FUNCTION_BLOCK FB_CheckAnyMode
VAR_INPUT
	
stn1:FB_Mode;
stn2:FB_Mode;
stn3:FB_Mode;
stn4:FB_Mode;
stn5:FB_Mode;
stn6:FB_Mode;


END_VAR
VAR_OUTPUT
	LockedModes:typeStationLockModes;
END_VAR
VAR
	tAnyAutoMode: BOOL;
	tAnyManualMode: BOOL;
END_VAR

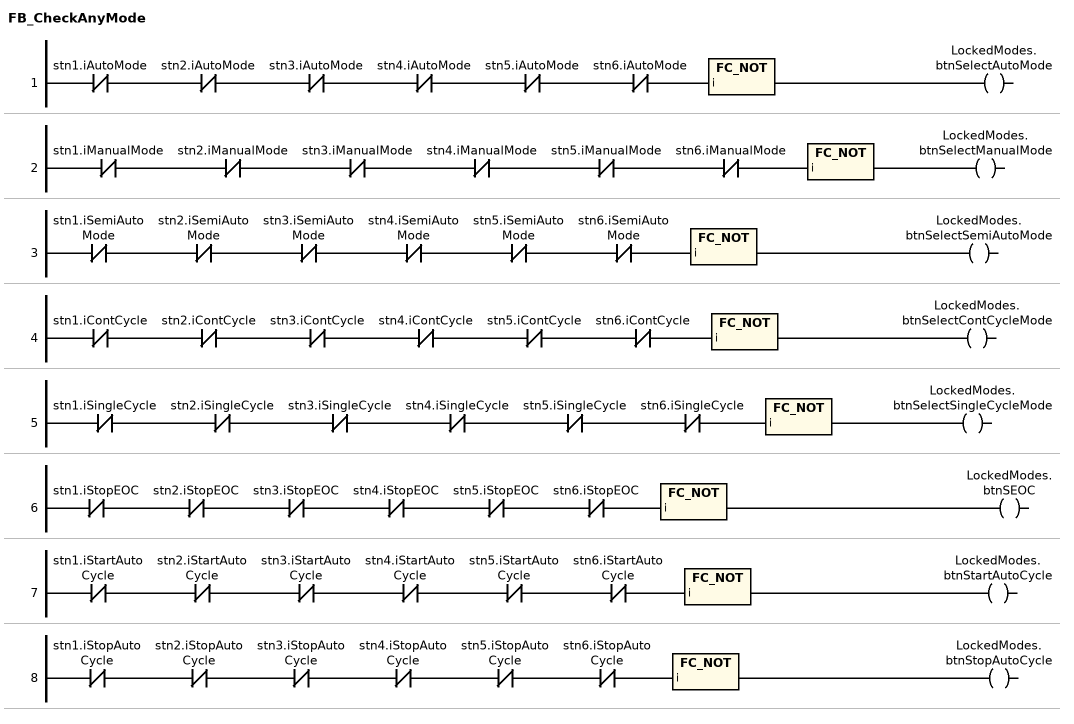
// NETWORK 1
LockedModes.btnSelectAutoMode := FC_NOT(i := NOT stn1.iAutoMode AND NOT stn2.iAutoMode AND NOT stn3.iAutoMode AND NOT stn4.iAutoMode AND NOT stn5.iAutoMode AND NOT stn6.iAutoMode);

// NETWORK 2
LockedModes.btnSelectManualMode := FC_NOT(i := NOT stn1.iManualMode AND NOT stn2.iManualMode AND NOT stn3.iManualMode AND NOT stn4.iManualMode AND NOT stn5.iManualMode AND NOT stn6.iManualMode);

// NETWORK 3
LockedModes.btnSelectSemiAutoMode := FC_NOT(i := NOT stn1.iSemiAutoMode AND NOT stn2.iSemiAutoMode AND NOT stn3.iSemiAutoMode AND NOT stn4.iSemiAutoMode AND NOT stn5.iSemiAutoMode AND NOT stn6.iSemiAutoMode);

// NETWORK 4
LockedModes.btnSelectContCycleMode := FC_NOT(i := NOT stn1.iContCycle AND NOT stn2.iContCycle AND NOT stn3.iContCycle AND NOT stn4.iContCycle AND NOT stn5.iContCycle AND NOT stn6.iContCycle);

// NETWORK 5
LockedModes.btnSelectSingleCycleMode := FC_NOT(i := NOT stn1.iSingleCycle AND NOT stn2.iSingleCycle AND NOT stn3.iSingleCycle AND NOT stn4.iSingleCycle AND NOT stn5.iSingleCycle AND NOT stn6.iSingleCycle);

// NETWORK 6
LockedModes.btnSEOC := FC_NOT(i := NOT stn1.iStopEOC AND NOT stn2.iStopEOC AND NOT stn3.iStopEOC AND NOT stn4.iStopEOC AND NOT stn5.iStopEOC AND NOT stn6.iStopEOC);

// NETWORK 7
LockedModes.btnStartAutoCycle := FC_NOT(i := NOT stn1.iStartAutoCycle AND NOT stn2.iStartAutoCycle AND NOT stn3.iStartAutoCycle AND NOT stn4.iStartAutoCycle AND NOT stn5.iStartAutoCycle AND NOT stn6.iStartAutoCycle);

// NETWORK 8
LockedModes.btnStopAutoCycle := FC_NOT(i := NOT stn1.iStopAutoCycle AND NOT stn2.iStopAutoCycle AND NOT stn3.iStopAutoCycle AND NOT stn4.iStopAutoCycle AND NOT stn5.iStopAutoCycle AND NOT stn6.iStopAutoCycle);

END_FUNCTION_BLOCK

(* stored: Version 1.1.0.1, ProductVersion 3.1.4024.11
   POU FB_CheckAnyMode: Id {a8851fa1-d96b-0a47-0ca5-1e8453d982a9}, SpecialFunc None *)
